FUNCTION F_FindFactorial :ULINT
VAR_INPUT
	n:ULINT;
END_VAR
VAR
	nReturnValue: ULINT;
	i: ULINT;
END_VAR

nReturnValue:=1;
FOR i:=1 TO N BY 1 DO
	nReturnValue := nReturnValue*i;
END_FOR

F_FindFactorial := nReturnValue;

END_FUNCTION

(* stored: Version 1.1.0.1, ProductVersion 3.1.4024.16
   POU F_FindFactorial: Id {5900008b-b0c1-4291-8240-abad8845df2a}, SpecialFunc None *)
